% RSLogix 500 project INTRO TO PLC - JOB 15.RSS, saved by version 10.00.00.00 %
PROJECT "PL06B"    % processor: Bul.1763 MicroLogix 1100 Series B %

PROGRAM FILES
  LAD 2   8 rungs

DATA FILES
  O0 OUTPUT  4 elements
  I1 INPUT  6 elements
  S2 STATUS  66 elements
  B3 BINARY  1 elements
  T4 TIMER  3 elements
  C5 COUNTER  2 elements
  R6 CONTROL  1 elements
  N7 INTEGER  1 elements
  F8 FLOAT  1 elements

LADDER 2
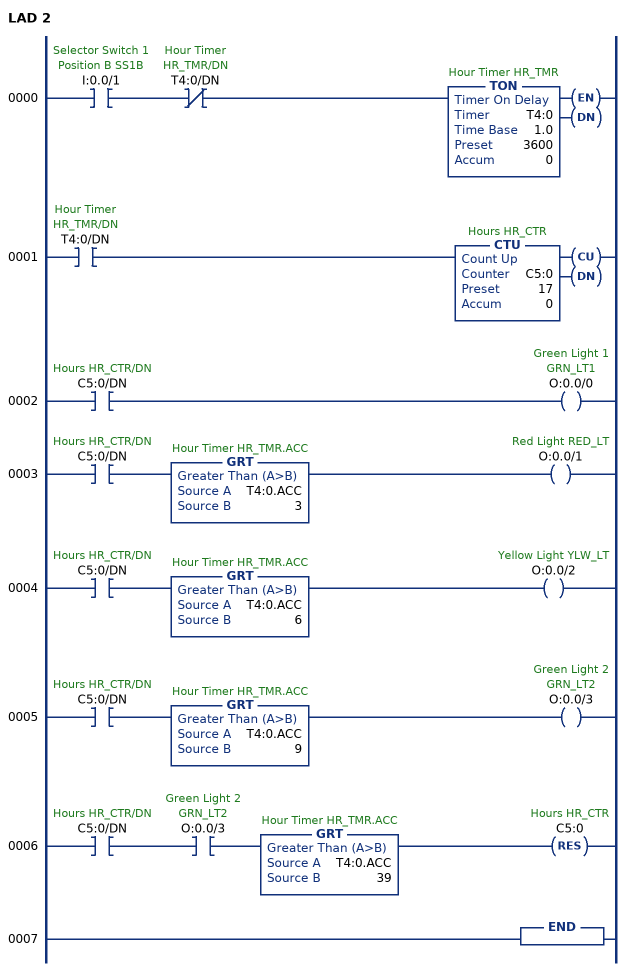
% Rung: 0 %
SOR XIC I:0.0/1 XIO T4:0/DN TON T4:0 1.0 3600 0 EOR
%   I:0.0/1  SS1B  "Selector Switch 1 Position B" %
%   T4:0  HR_TMR  "Hour Timer" %
% Rung: 1 %
SOR XIC T4:0/DN CTU C5:0 17 0 EOR
%   T4:0  HR_TMR  "Hour Timer" %
%   C5:0  HR_CTR  "Hours" %
% Rung: 2 %
SOR XIC C5:0/DN OTE O:0.0/0 EOR
%   C5:0  HR_CTR  "Hours" %
%   O:0.0/0  GRN_LT1  "Green Light 1" %
% Rung: 3 %
SOR XIC C5:0/DN GRT T4:0.ACC 3 OTE O:0.0/1 EOR
%   C5:0  HR_CTR  "Hours" %
%   T4:0  HR_TMR  "Hour Timer" %
%   O:0.0/1  RED_LT  "Red Light" %
% Rung: 4 %
SOR XIC C5:0/DN GRT T4:0.ACC 6 OTE O:0.0/2 EOR
%   C5:0  HR_CTR  "Hours" %
%   T4:0  HR_TMR  "Hour Timer" %
%   O:0.0/2  YLW_LT  "Yellow Light" %
% Rung: 5 %
SOR XIC C5:0/DN GRT T4:0.ACC 9 OTE O:0.0/3 EOR
%   C5:0  HR_CTR  "Hours" %
%   T4:0  HR_TMR  "Hour Timer" %
%   O:0.0/3  GRN_LT2  "Green Light 2" %
% Rung: 6 %
SOR XIC C5:0/DN XIC O:0.0/3 GRT T4:0.ACC 39 RES C5:0 EOR
%   C5:0  HR_CTR  "Hours" %
%   O:0.0/3  GRN_LT2  "Green Light 2" %
%   T4:0  HR_TMR  "Hour Timer" %
% Rung: 7 %
SOR END EOR

OTHER DOCUMENTED ADDRESSES
  B3:0/0  SEAL1  "Seal 1"
  B3:0/1  SEAL2  "Seal 2"
  B3:0/15  SCRATCH  "Scratch Bit"
  C5:1  HOUR_CTR  "Cycle Counter 2"
  I:0.0/0  SS1A  "Selector Switch 1 Position A"
  I:0.0/2  SS2A  "Selector Switch 2 Position A"
  I:0.0/3  SS2B  "Selector Switch 2 Position B"
  I:0.0/4  PB1  "Pushbutton 1"
  I:0.0/5  PB2  "Pushbutton 2"
  RTC:0.YR  RTC
  SEL1B  
  T4:1  INT_TMR  "Interval Timer"
  T4:2  RST_TMR  "Reset Timer"

DATA TABLE (non-zero values as saved)
DATA B3
% B3:0 % 0X800A
DATA T4
% .PRE .ACC %
% T4:0 % 3600 0
% T4:1 % 3 0
% T4:2 % 30 0
DATA C5
% .PRE .ACC %
% C5:0 % 17 0
% C5:1 % 16 0
